// TIA Portal V17 export
// export: Created 2024-08-09T12:52:13.9620512Z, ExportSetting WithDefaults, DisplayName Totally Integrated Automation Portal, DisplayVersion V17 Update 7, DisplayName TIA Portal Openness, DisplayVersion V17 Update 7, DisplayName TIA Portal Version Control Interface, DisplayVersion V17, DisplayName STEP 7 Professional, DisplayVersion V17 Update 7, DisplayName STEP 7 Safety, DisplayVersion V17 Update 6, DisplayName WinCC Professional, DisplayVersion V17 Update 7
DATA_BLOCK "DB_ChPont"   // DB30
{ S7_Optimized_Access := 'TRUE' }
VERSION : 0.1
// stored: AutoNumber true, DBAccessibleFromOPCUA true, DBAccessibleFromWebserver true, IsOnlyStoredInLoadMemory false, IsRetainMemResEnabled false, IsWriteProtectedInAS false, MemoryReserve 100
   VAR RETAIN
      ChPont { S7_SetPoint := 'True'} : Array[0..1] of "S_ChargPont";
   END_VAR
   VAR
      RazPtzs { ExternalAccessible := 'False'; ExternalVisible := 'False'; ExternalWritable := 'False'} : "S_SuiviCommande";
   END_VAR
BEGIN
END_DATA_BLOCK
